# EPICS autosave request: iocBoot/iocTomoScanStream_2BMB/auto_settings.req
file "tomoScan_settings.req", P=$(P), R=$(R)
file "tomoScan_PSO_settings.req", P=$(P), R=$(R)
file "tomoScan_2BM_settings.req", P=$(P), R=$(R)
file "tomoScanStream_settings.req", P=$(P), R=$(R)
